PROGRAM MAIN
VAR
	// TcUnit finds every FB_TestSuite instance by itself; it is enough to declare them here.
	fbCoverControlTests	: FB_MonetCoverControl_Tests;
	fbAzimuthOffsetTests	: F_AzimuthOffsetOnAxis_Tests;
END_VAR

TcUnit.RUN();

END_PROGRAM

(* stored: Version 1.1.0.1, ProductVersion 3.1.4024.15
   POU MAIN: Id {0799da45-8949-418f-b539-2af88eaf4ab8}, SpecialFunc None *)
